// TIA Portal V19 export
DATA_BLOCK "MGF AUTO DB"   // DB57
{ S7_Optimized_Access := 'FALSE' }
   VAR RETAIN
      OUTPUT : Struct
         "NAOCL DOSING" : Bool;
      END_STRUCT;
      "MGF SERVIC _TIMER SET" : Int;
      "MGF SERVIC _TIMER PV" : Int;
      "BACKWASH_TIMER SET" : Int;
      "BACKWASH_TIMER PV" : Int;
      "RINSE MODE TIMER SET" : Int;
      "RINSE MODE TIMER PV" : Int;
   END_VAR
BEGIN
END_DATA_BLOCK
